FUNCTION_BLOCK FB_Abfuellmodul
VAR_INPUT
	bEnable : BOOL;
	bExecute : BOOL;
	nstation : INT;
 		
END_VAR
VAR_OUTPUT
	estate : eBetriebszustand;
END_VAR
VAR
	fbVereinzelung : FB_Vereinzelung;
	fbTransport : FB_Transport;
	fbDispenser1 : FB_Dispenser;
	fbDispenser2 : FB_Dispenser;
	fbDispenser3 : FB_Dispenser;
	nstate : INT := 100;
END_VAR

CASE nstate OF 
	0: // Off
	fbVereinzelung.benable := FALSE;
	fbTransport.bEnable := FALSE;
	fbDispenser1.bEnable := FALSE;
	fbDispenser2.bEnable := FALSE;
	fbDispenser3.bEnable := FALSE;
	
	
	fbVereinzelung.bexecute := FALSE;
	fbTransport.bExecute := FALSE;
	fbDispenser1.bExecute := FALSE;
	fbDispenser2.bExecute := FALSE;
	fbDispenser3.bExecute := FALSE;
	
	eState :=eBetriebszustand.off;
	
	IF bEnable THEN
		nstate := 10; // Init
	END_IF
	
	10: // Init
	fbVereinzelung.benable := TRUE;
	fbTransport.bEnable := TRUE;
	fbDispenser1.bEnable := TRUE;
	fbDispenser2.bEnable := TRUE;
	fbDispenser3.bEnable := TRUE;
	
	
	fbVereinzelung.bexecute := FALSE;
	fbTransport.bExecute := FALSE;
	fbDispenser1.bExecute := FALSE;
	fbDispenser2.bExecute := FALSE;
	fbDispenser3.bExecute := FALSE;
	
	eState :=eBetriebszustand.init;
	
	IF fbVereinzelung.estate = eBetriebszustand.ready AND 
		fbVereinzelung.estate = eBetriebszustand.ready THEN
		nstate := 20; // Ready
	END_IF
	
	20: // Ready
	fbVereinzelung.benable := TRUE;
	fbTransport.bEnable := TRUE;
	fbDispenser1.bEnable := TRUE;
	fbDispenser2.bEnable := TRUE;
	fbDispenser3.bEnable := TRUE;
	
	IF bExecute THEN
		nState := 30; // Start
	END_IF
	
	30: // Start
	fbVereinzelung.bExecute := TRUE;
	fbTransport.bExecute := TRUE;
	fbDispenser1.bExecute := FALSE;
	fbDispenser2.bExecute := FALSE;
	fbDispenser3.bExecute := FALSE;
	
	eState := eBetriebszustand.Production;
	
	nStation := 1;

	IF fbVereinzelung.estate = eBetriebszustand.done AND 
		fbTransport.eState = eBetriebszustand.done THEN
		nstate := 31; // Extruder 1
	END_IF
		
	31: // Extruder 1
	nStation := 1;
	fbDispenser1.bExecute := TRUE;
	fbDispenser2.bExecute := FALSE;
	fbDispenser3.bExecute := FALSE;
	
	IF fbDispenser1.estate = eBetriebszustand.Done THEN 
		nstate := 32; // Bewegung zu 2.Station
	END_IF
		
	32:// Bewegung zu 2.Station
	nStation := 2;
	fbTransport.bExecute := TRUE;
	fbDispenser1.bExecute := FALSE;
	fbDispenser2.bExecute := FALSE;
	fbDispenser3.bExecute := FALSE;
	
	IF fbTransport.eState = eBetriebszustand.done THEN
		nState := 33; // zweiter Extruder
	END_IF
	
	33: // zweiter Extruder
	nStation := 2
	fbDispenser2.bExecute := TRUE;

	IF fbDispenser2.eState = eBetriebszustand.Done THEN 
		nstate := 34; // Bewegung zu 3.Station
	END_IF
	
	34: // Bewegung zu 3.Station
	nStation := 3;
	fbTransport.bExecute := TRUE;
	fbDispenser1.bExecute := FALSE;
	fbDispenser2.bExecute := FALSE;
	fbDispenser3.bExecute := FALSE;
	
	IF fbTransport.eState = eBetriebszustand.done THEN
		nState := 35; // Extruder 3
	END_IF
	
	35: // Extruder 3
	nStation := 3;
	fbDispenser1.bExecute := FALSE;
	fbDispenser2.bExecute := FALSE;
	fbDispenser3.bExecute := TRUE;
	
	IF fbDispenser3.estate = eBetriebszustand.done THEN
		nState := 36; // Bewegung zu Ende
	END_IF
	
	36: // Bewegung zu Ende
	nStation := 4;
	fbTransport.bExecute := TRUE;
	fbDispenser1.bExecute := FALSE;
	fbDispenser2.bExecute := FALSE;
	fbDispenser3.bExecute := FALSE;
	
	IF fbTransport.eState = eBetriebszustand.done THEN
		nState := 40; //Done
	END_IF
	
	40: // Done
	
	estate:= eBetriebszustand.done;
	
	fbTransport.bExecute := FALSE;
	fbDispenser1.bExecute := FALSE;
	fbDispenser2.bExecute := FALSE;
	fbDispenser3.bExecute := FALSE;
	
	
	
END_CASE

END_FUNCTION_BLOCK

(* stored: Version 1.1.0.1, ProductVersion 3.1.4024.15
   POU FB_Abfuellmodul: Id {735a87f2-dd00-4b8e-8fa6-60d88a866885}, SpecialFunc None *)
